COMM SMOVL C00306 BC00306 V=60.0  +MOVJ EC00306
COMM SMOVL C00307 BC00307 V=60.0  +MOVJ EC00307
COMM SREFP 3 C00308 BC00308  +REFP EC00308
COMM CALL JOB:SEARCH-R1-S13D
COMM SET P041 P006
COMM SFTON3D P041
COMM SMOVL C00309 BC00309 V=60.0  +MOVJ EC00309
COMM MOVL C00310 BC00310 V=400.0  +MOVJ EC00310 VJ=100.00
COMM MOVL C00311 BC00311 V=1000.0  +MOVJ EC00311 VJ=100.00
COMM 'Path S1858
COMM SFTOF3D
COMM MOVJ C00312 BC00312 VJ=100.00  +MOVJ EC00312 VJ=100.00
COMM MOVL C00313 BC00313 V=400.0  +MOVJ EC00313 VJ=100.00
COMM SMOVL C00314 BC00314 V=60.0  +MOVJ EC00314
COMM SREFP 3 C00315 BC00315  +REFP EC00315
COMM CALL JOB:SEARCH-R1-S13D
COMM SET P040 P006
COMM SFTON3D P040
COMM SMOVL C00316 BC00316 V=60.0  +MOVJ EC00316
COMM SMOVL C00317 BC00317 V=60.0  +MOVJ EC00317
COMM SREFP 3 C00318 BC00318  +REFP EC00318
COMM CALL JOB:SEARCH-R1-S13D
COMM SET P040 P006
COMM SFTON3D P040
COMM SMOVL C00319 BC00319 V=60.0  +MOVJ EC00319
COMM MOVL C00320 BC00320 V=400.0  +MOVJ EC00320 VJ=100.00
COMM MOVL C00321 BC00321 V=1000.0  +MOVJ EC00321 VJ=100.00
MOVL C00322 BC00322 V=1000.0  +MOVJ EC00322 VJ=100.00
'Path S1859
SFTOF3D
MOVJ C00323 BC00323 VJ=100.00  +MOVJ EC00323 VJ=100.00
MOVJ C00324 BC00324 VJ=100.00  +MOVJ EC00324 VJ=100.00
MOVL C00325 BC00325 V=400.0  +MOVJ EC00325 VJ=100.00
SMOVL C00326 BC00326 V=60.0  +MOVJ EC00326
SREFP 3 C00327 BC00327  +REFP EC00327
CALL JOB:SEARCH-R1-S13D
SET P043 P006
SFTON3D P043
SMOVL C00328 BC00328 V=60.0  +MOVJ EC00328
SMOVL C00329 BC00329 V=60.0  +MOVJ EC00329
SREFP 3 C00330 BC00330  +REFP EC00330
CALL JOB:SEARCH-R1-S13D
SET P043 P006
SFTON3D P043
SMOVL C00331 BC00331 V=60.0  +MOVJ EC00331
MOVL C00332 BC00332 V=400.0  +MOVJ EC00332 VJ=100.00
MOVL C00333 BC00333 V=1000.0  +MOVJ EC00333 VJ=100.00
'Path S1860
SFTOF3D
MOVJ C00334 BC00334 VJ=100.00  +MOVJ EC00334 VJ=100.00
MOVL C00335 BC00335 V=400.0  +MOVJ EC00335 VJ=100.00
SMOVL C00336 BC00336 V=60.0  +MOVJ EC00336
SREFP 3 C00337 BC00337  +REFP EC00337
CALL JOB:SEARCH-R1-S13D
SET P039 P006
SFTON3D P039
SMOVL C00338 BC00338 V=60.0  +MOVJ EC00338
SMOVL C00339 BC00339 V=60.0  +MOVJ EC00339
SREFP 3 C00340 BC00340  +REFP EC00340
CALL JOB:SEARCH-R1-S13D
SET P039 P006
SFTON3D P039
SMOVL C00341 BC00341 V=60.0  +MOVJ EC00341
MOVL C00342 BC00342 V=400.0  +MOVJ EC00342 VJ=100.00
MOVL C00343 BC00343 V=1000.0  +MOVJ EC00343 VJ=100.00
MOVJ C00344 BC00344 VJ=100.00  +MOVJ EC00344 VJ=100.00
'Path S1861
SFTOF3D
MOVJ C00345 BC00345 VJ=100.00  +MOVJ EC00345 VJ=100.00
MOVL C00346 BC00346 V=400.0  +MOVJ EC00346 VJ=100.00
SMOVL C00347 BC00347 V=60.0  +MOVJ EC00347
SREFP 3 C00348 BC00348  +REFP EC00348
CALL JOB:SEARCH-R1-S13D
SET P034 P006
SFTON3D P034
SMOVL C00349 BC00349 V=60.0  +MOVJ EC00349
SMOVL C00350 BC00350 V=60.0  +MOVJ EC00350
SREFP 3 C00351 BC00351  +REFP EC00351
CALL JOB:SEARCH-R1-S13D
SET P034 P006
SFTON3D P034
SMOVL C00352 BC00352 V=60.0  +MOVJ EC00352
MOVL C00353 BC00353 V=400.0  +MOVJ EC00353 VJ=100.00
MOVL C00354 BC00354 V=1000.0  +MOVJ EC00354 VJ=100.00
MOVJ C00355 BC00355 VJ=100.00  +MOVJ EC00355 VJ=100.00
'Path S1862
SFTOF3D
MOVJ C00356 BC00356 VJ=100.00  +MOVJ EC00356 VJ=100.00
MOVL C00357 BC00357 V=400.0  +MOVJ EC00357 VJ=100.00
SMOVL C00358 BC00358 V=60.0  +MOVJ EC00358
SREFP 3 C00359 BC00359  +REFP EC00359
CALL JOB:SEARCH-R1-S13D
SET P038 P006
SFTON3D P038
SMOVL C00360 BC00360 V=60.0  +MOVJ EC00360
SMOVL C00361 BC00361 V=60.0  +MOVJ EC00361
SREFP 3 C00362 BC00362  +REFP EC00362
CALL JOB:SEARCH-R1-S13D
SET P038 P006
SFTON3D P038
SMOVL C00363 BC00363 V=60.0  +MOVJ EC00363
SMOVL C00364 BC00364 V=60.0  +MOVJ EC00364
SREFP 3 C00365 BC00365  +REFP EC00365
CALL JOB:SEARCH-R1-S13D
SET P038 P006
SFTON3D P038
SMOVL C00366 BC00366 V=60.0  +MOVJ EC00366
MOVL C00367 BC00367 V=400.0  +MOVJ EC00367 VJ=100.00
MOVL C00368 BC00368 V=1000.0  +MOVJ EC00368 VJ=100.00
'Path S1863
SFTOF3D
MOVJ C00369 BC00369 VJ=100.00  +MOVJ EC00369 VJ=100.00
MOVL C00370 BC00370 V=400.0  +MOVJ EC00370 VJ=100.00
SMOVL C00371 BC00371 V=60.0  +MOVJ EC00371
SREFP 3 C00372 BC00372  +REFP EC00372
CALL JOB:SEARCH-R1-S13D
SET P033 P006
SFTON3D P033
SMOVL C00373 BC00373 V=60.0  +MOVJ EC00373
SMOVL C00374 BC00374 V=60.0  +MOVJ EC00374
SREFP 3 C00375 BC00375  +REFP EC00375
CALL JOB:SEARCH-R1-S13D
SET P033 P006
SFTON3D P033
SMOVL C00376 BC00376 V=60.0  +MOVJ EC00376
MOVL C00377 BC00377 V=400.0  +MOVJ EC00377 VJ=100.00
MOVL C00378 BC00378 V=1000.0  +MOVJ EC00378 VJ=100.00
MOVL C00379 BC00379 V=1000.0  +MOVJ EC00379 VJ=100.00
'Path S1864
SFTOF3D
MOVJ C00380 BC00380 VJ=100.00  +MOVJ EC00380 VJ=100.00
MOVJ C00381 BC00381 VJ=100.00  +MOVJ EC00381 VJ=100.00
MOVL C00382 BC00382 V=400.0  +MOVJ EC00382 VJ=100.00
SMOVL C00383 BC00383 V=60.0  +MOVJ EC00383
SREFP 3 C00384 BC00384  +REFP EC00384
CALL JOB:SEARCH-R1-S13D
SET P035 P006
SFTON3D P035
SMOVL C00385 BC00385 V=60.0  +MOVJ EC00385
SMOVL C00386 BC00386 V=60.0  +MOVJ EC00386
SREFP 3 C00387 BC00387  +REFP EC00387
CALL JOB:SEARCH-R1-S13D
SET P035 P006
SFTON3D P035
SMOVL C00388 BC00388 V=60.0  +MOVJ EC00388
MOVL C00389 BC00389 V=400.0  +MOVJ EC00389 VJ=100.00
MOVL C00390 BC00390 V=1000.0  +MOVJ EC00390 VJ=100.00
MOVL C00391 BC00391 V=1000.0  +MOVJ EC00391 VJ=100.00
'Path S1865
SFTOF3D
MOVJ C00392 BC00392 VJ=100.00  +MOVJ EC00392 VJ=100.00
MOVL C00393 BC00393 V=400.0  +MOVJ EC00393 VJ=100.00
SMOVL C00394 BC00394 V=60.0  +MOVJ EC00394
SREFP 3 C00395 BC00395  +REFP EC00395
CALL JOB:SEARCH-R1-S13D
SET P037 P006
SFTON3D P037
SMOVL C00396 BC00396 V=60.0  +MOVJ EC00396
SMOVL C00397 BC00397 V=60.0  +MOVJ EC00397
SREFP 3 C00398 BC00398  +REFP EC00398
CALL JOB:SEARCH-R1-S13D
SET P037 P006
SFTON3D P037
SMOVL C00399 BC00399 V=60.0  +MOVJ EC00399
MOVL C00400 BC00400 V=400.0  +MOVJ EC00400 VJ=100.00
MOVL C00401 BC00401 V=1000.0  +MOVJ EC00401 VJ=100.00
'Path S1866
SFTOF3D
MOVJ C00402 BC00402 VJ=100.00  +MOVJ EC00402 VJ=100.00
MOVJ C00403 BC00403 VJ=100.00  +MOVJ EC00403 VJ=100.00
MOVL C00404 BC00404 V=400.0  +MOVJ EC00404 VJ=100.00
SMOVL C00405 BC00405 V=60.0  +MOVJ EC00405
SREFP 3 C00406 BC00406  +REFP EC00406
CALL JOB:SEARCH-R1-S13D
SET P031 P006
SFTON3D P031
SMOVL C00407 BC00407 V=60.0  +MOVJ EC00407
SMOVL C00408 BC00408 V=60.0  +MOVJ EC00408
SREFP 3 C00409 BC00409  +REFP EC00409
CALL JOB:SEARCH-R1-S13D
SET P031 P006
SFTON3D P031
SMOVL C00410 BC00410 V=60.0  +MOVJ EC00410
MOVL C00411 BC00411 V=400.0  +MOVJ EC00411 VJ=100.00
MOVL C00412 BC00412 V=1000.0  +MOVJ EC00412 VJ=100.00
'Path S1867
MOVJ C00413 BC00413 VJ=20.00  +MOVJ EC00413 VJ=20.00
MOVJ C00414 BC00414 VJ=20.00  +MOVJ EC00414 VJ=20.00
SFTOF3D
MOVJ C00415 BC00415 VJ=100.00  +MOVJ EC00415 VJ=100.00
MOVL C00416 BC00416 V=400.0  +MOVJ EC00416 VJ=100.00
SMOVL C00417 BC00417 V=60.0  +MOVJ EC00417
SREFP 3 C00418 BC00418  +REFP EC00418
CALL JOB:SEARCH-R1-S13D
SET P036 P006
SFTON3D P036
SMOVL C00419 BC00419 V=60.0  +MOVJ EC00419
SMOVL C00420 BC00420 V=60.0  +MOVJ EC00420
SREFP 3 C00421 BC00421  +REFP EC00421
CALL JOB:SEARCH-R1-S13D
SET P036 P006
SFTON3D P036
SMOVL C00422 BC00422 V=60.0  +MOVJ EC00422
MOVL C00423 BC00423 V=400.0  +MOVJ EC00423 VJ=100.00
MOVL C00424 BC00424 V=1000.0  +MOVJ EC00424 VJ=100.00
MOVL C00425 BC00425 V=1000.0  +MOVJ EC00425 VJ=100.00
'Path S1868
SFTOF3D
MOVJ C00426 BC00426 VJ=100.00  +MOVJ EC00426 VJ=100.00
MOVL C00427 BC00427 V=400.0  +MOVJ EC00427 VJ=100.00
SMOVL C00428 BC00428 V=60.0  +MOVJ EC00428
SREFP 3 C00429 BC00429  +REFP EC00429
CALL JOB:SEARCH-R1-S13D
SET P032 P006
SFTON3D P032
SMOVL C00430 BC00430 V=60.0  +MOVJ EC00430
SMOVL C00431 BC00431 V=60.0  +MOVJ EC00431
SREFP 3 C00432 BC00432  +REFP EC00432
CALL JOB:SEARCH-R1-S13D
SET P032 P006
SFTON3D P032
SMOVL C00433 BC00433 V=60.0  +MOVJ EC00433
MOVL C00434 BC00434 V=400.0  +MOVJ EC00434 VJ=100.00
MOVL C00435 BC00435 V=1000.0  +MOVJ EC00435 VJ=100.00
'Path W1869
SFTOF3D
SFTON3D P032
MOVJ C00436 BC00436 VJ=100.00  +MOVJ EC00436 VJ=100.00
SMOVL C00437 BC00437 V=400.0  +MOVJ EC00437
SMOVL C00438 BC00438 V=100.0 PL=0  +MOVJ EC00438
SREFP 1 C00439 BC00439  +REFP EC00439
SREFP 2 C00440 BC00440  +REFP EC00440
MACRO1 MJ#(0) ARGF0
ARCON
SMOVL C00441 BC00441 V=10.0  +MOVJ EC00441
SMOVL C00442 BC00442 V=10.0  +MOVJ EC00442
SMOVL C00443 BC00443 V=10.0  +MOVJ EC00443
ARCOF
SMOVL C00444 BC00444 V=400.0  +MOVJ EC00444
SMOVL C00445 BC00445 V=1000.0  +MOVJ EC00445
SMOVL C00446 BC00446 V=1000.0  +MOVJ EC00446
SFTOF3D
MOVJ C00447 BC00447 VJ=100.00  +MOVJ EC00447 VJ=100.00
'Path W1870
SFTOF3D
SFTON3D P033
MOVJ C00448 BC00448 VJ=100.00  +MOVJ EC00448 VJ=100.00
MOVJ C00449 BC00449 VJ=100.00  +MOVJ EC00449 VJ=100.00
SMOVL C00450 BC00450 V=400.0  +MOVJ EC00450
SMOVL C00451 BC00451 V=100.0 PL=0  +MOVJ EC00451
SREFP 1 C00452 BC00452  +REFP EC00452
SREFP 2 C00453 BC00453  +REFP EC00453
MACRO1 MJ#(0) ARGF0
ARCON
SMOVL C00454 BC00454 V=10.0  +MOVJ EC00454
SMOVL C00455 BC00455 V=10.0  +MOVJ EC00455
SMOVL C00456 BC00456 V=10.0  +MOVJ EC00456
ARCOF
SMOVL C00457 BC00457 V=400.0  +MOVJ EC00457
SMOVL C00458 BC00458 V=1000.0  +MOVJ EC00458
SFTOF3D
'Path W1871
SFTOF3D
SFTON3D P034
MOVJ C00459 BC00459 VJ=100.00  +MOVJ EC00459 VJ=100.00
SMOVL C00460 BC00460 V=400.0  +MOVJ EC00460
SMOVL C00461 BC00461 V=100.0 PL=0  +MOVJ EC00461
SREFP 1 C00462 BC00462  +REFP EC00462
SREFP 2 C00463 BC00463  +REFP EC00463
MACRO1 MJ#(0) ARGF0
ARCON
SMOVL C00464 BC00464 V=10.0  +MOVJ EC00464
SMOVL C00465 BC00465 V=10.0  +MOVJ EC00465
ARCOF
SMOVL C00466 BC00466 V=400.0  +MOVJ EC00466
SMOVL C00467 BC00467 V=1000.0  +MOVJ EC00467
SMOVL C00468 BC00468 V=1000.0  +MOVJ EC00468
SFTOF3D
MOVJ C00469 BC00469 VJ=20.00  +MOVJ EC00469 VJ=20.00
MOVJ C00470 BC00470 VJ=20.00  +MOVJ EC00470 VJ=20.00
'Path W1872
SFTOF3D
SFTON3D P031
MOVJ C00471 BC00471 VJ=100.00  +MOVJ EC00471 VJ=100.00
SMOVL C00472 BC00472 V=400.0  +MOVJ EC00472
SMOVL C00473 BC00473 V=100.0 PL=0  +MOVJ EC00473
SREFP 1 C00474 BC00474  +REFP EC00474
SREFP 2 C00475 BC00475  +REFP EC00475
MACRO1 MJ#(0) ARGF0
ARCON
SMOVL C00476 BC00476 V=10.0  +MOVJ EC00476
SMOVL C00477 BC00477 V=10.0  +MOVJ EC00477
ARCOF
SMOVL C00478 BC00478 V=400.0  +MOVJ EC00478
SMOVL C00479 BC00479 V=1000.0  +MOVJ EC00479
SMOVL C00480 BC00480 V=1000.0  +MOVJ EC00480
SFTOF3D
'Path W1873
MOVJ C00481 BC00481 VJ=20.00  +MOVJ EC00481 VJ=20.00
SFTOF3D
SFTON3D P035
MOVJ C00482 BC00482 VJ=100.00  +MOVJ EC00482 VJ=100.00
SMOVL C00483 BC00483 V=400.0  +MOVJ EC00483
SMOVL C00484 BC00484 V=100.0 PL=0  +MOVJ EC00484
SREFP 1 C00485 BC00485  +REFP EC00485
SREFP 2 C00486 BC00486  +REFP EC00486
MACRO1 MJ#(0) ARGF0
ARCON
SMOVL C00487 BC00487 V=10.0  +MOVJ EC00487
SMOVL C00488 BC00488 V=10.0  +MOVJ EC00488
ARCOF
SMOVL C00489 BC00489 V=400.0  +MOVJ EC00489
SMOVL C00490 BC00490 V=1000.0  +MOVJ EC00490
SMOVL C00491 BC00491 V=1000.0  +MOVJ EC00491
SFTOF3D
MOVJ C00492 BC00492 VJ=100.00  +MOVJ EC00492 VJ=100.00
'Path W1874
SFTOF3D
SFTON3D P036
MOVJ C00493 BC00493 VJ=100.00  +MOVJ EC00493 VJ=100.00
SMOVL C00494 BC00494 V=400.0  +MOVJ EC00494
SMOVL C00495 BC00495 V=100.0 PL=0  +MOVJ EC00495
SREFP 1 C00496 BC00496  +REFP EC00496
SREFP 2 C00497 BC00497  +REFP EC00497
MACRO1 MJ#(0) ARGF0
ARCON
SMOVL C00498 BC00498 V=10.0  +MOVJ EC00498
SMOVL C00499 BC00499 V=10.0  +MOVJ EC00499
SMOVL C00500 BC00500 V=10.0  +MOVJ EC00500
ARCOF
SMOVL C00501 BC00501 V=400.0  +MOVJ EC00501
SMOVL C00502 BC00502 V=1000.0  +MOVJ EC00502
SMOVL C00503 BC00503 V=1000.0  +MOVJ EC00503
SFTOF3D
MOVJ C00504 BC00504 VJ=100.00  +MOVJ EC00504 VJ=100.00
'Path W1875
SFTOF3D
SFTON3D P037
MOVJ C00505 BC00505 VJ=100.00  +MOVJ EC00505 VJ=100.00
MOVJ C00506 BC00506 VJ=100.00  +MOVJ EC00506 VJ=100.00
SMOVL C00507 BC00507 V=400.0  +MOVJ EC00507
SMOVL C00508 BC00508 V=100.0 PL=0  +MOVJ EC00508
SREFP 1 C00509 BC00509  +REFP EC00509
SREFP 2 C00510 BC00510  +REFP EC00510
MACRO1 MJ#(0) ARGF0
ARCON
SMOVL C00511 BC00511 V=10.0  +MOVJ EC00511
SMOVL C00512 BC00512 V=10.0  +MOVJ EC00512
SMOVL C00513 BC00513 V=10.0  +MOVJ EC00513
ARCOF
SMOVL C00514 BC00514 V=400.0  +MOVJ EC00514
SMOVL C00515 BC00515 V=1000.0  +MOVJ EC00515
SMOVL C00516 BC00516 V=1000.0  +MOVJ EC00516
SFTOF3D
MOVJ C00517 BC00517 VJ=100.00  +MOVJ EC00517 VJ=100.00
'Path W1876
SFTOF3D
SFTON3D P038
MOVJ C00518 BC00518 VJ=100.00  +MOVJ EC00518 VJ=100.00
MOVJ C00519 BC00519 VJ=100.00  +MOVJ EC00519 VJ=100.00
SMOVL C00520 BC00520 V=400.0  +MOVJ EC00520
SMOVL C00521 BC00521 V=100.0 PL=0  +MOVJ EC00521
SREFP 1 C00522 BC00522  +REFP EC00522
SREFP 2 C00523 BC00523  +REFP EC00523
MACRO1 MJ#(0) ARGF0
ARCON
SMOVL C00524 BC00524 V=10.0  +MOVJ EC00524
SMOVL C00525 BC00525 V=10.0  +MOVJ EC00525
ARCOF
SMOVL C00526 BC00526 V=400.0  +MOVJ EC00526
SMOVL C00527 BC00527 V=1000.0  +MOVJ EC00527
SFTOF3D
'Path W1877
SFTOF3D
SFTON3D P038
SMOVL C00528 BC00528 V=400.0  +MOVJ EC00528
SMOVL C00529 BC00529 V=100.0 PL=0  +MOVJ EC00529
SREFP 1 C00530 BC00530  +REFP EC00530
SREFP 2 C00531 BC00531  +REFP EC00531
MACRO1 MJ#(0) ARGF0
ARCON
SMOVL C00532 BC00532 V=10.0  +MOVJ EC00532
SMOVL C00533 BC00533 V=10.0  +MOVJ EC00533
SMOVL C00534 BC00534 V=10.0  +MOVJ EC00534
ARCOF
SMOVL C00535 BC00535 V=400.0  +MOVJ EC00535
SFTOF3D
MOVJ C00536 BC00536 VJ=100.00  +MOVJ EC00536 VJ=100.00
'Path W1878
SFTOF3D
SFTON3D P039
MOVJ C00537 BC00537 VJ=100.00  +MOVJ EC00537 VJ=100.00
MOVJ C00538 BC00538 VJ=100.00  +MOVJ EC00538 VJ=100.00
SMOVL C00539 BC00539 V=400.0  +MOVJ EC00539
SMOVL C00540 BC00540 V=100.0 PL=0  +MOVJ EC00540
SREFP 1 C00541 BC00541  +REFP EC00541
SREFP 2 C00542 BC00542  +REFP EC00542
MACRO1 MJ#(0) ARGF0
ARCON
SMOVL C00543 BC00543 V=10.0  +MOVJ EC00543
ARCOF
SMOVL C00544 BC00544 V=400.0  +MOVJ EC00544
SMOVL C00545 BC00545 V=1000.0  +MOVJ EC00545
SMOVL C00546 BC00546 V=1000.0  +MOVJ EC00546
SFTOF3D
'Path W1879
SFTOF3D
SFTON3D P042
MOVJ C00547 BC00547 VJ=100.00  +MOVJ EC00547 VJ=100.00
COMM MOVJ C00548 BC00548 VJ=100.00  +MOVJ EC00548 VJ=100.00
COMM SMOVL C00549 BC00549 V=400.0  +MOVJ EC00549
COMM SMOVL C00550 BC00550 V=100.0 PL=0  +MOVJ EC00550
COMM SREFP 1 C00551 BC00551  +REFP EC00551
COMM SREFP 2 C00552 BC00552  +REFP EC00552
COMM MACRO1 MJ#(0) ARGF0
COMM ARCON
COMM SMOVL C00553 BC00553 V=10.0  +MOVJ EC00553
COMM SMOVL C00554 BC00554 V=10.0  +MOVJ EC00554
COMM SMOVL C00555 BC00555 V=10.0  +MOVJ EC00555
COMM ARCOF
COMM SMOVL C00556 BC00556 V=400.0  +MOVJ EC00556
COMM SMOVL C00557 BC00557 V=1000.0  +MOVJ EC00557
SFTOF3D
'Path W1880
COMM SFTOF3D
COMM SFTON3D P041
COMM MOVJ C00558 BC00558 VJ=100.00  +MOVJ EC00558 VJ=100.00
COMM SMOVL C00559 BC00559 V=400.0  +MOVJ EC00559
COMM SMOVL C00560 BC00560 V=100.0 PL=0  +MOVJ EC00560
COMM SREFP 1 C00561 BC00561  +REFP EC00561
COMM SREFP 2 C00562 BC00562  +REFP EC00562
COMM MACRO1 MJ#(0) ARGF0
COMM ARCON
COMM SMOVL C00563 BC00563 V=10.0  +MOVJ EC00563
COMM ARCOF
COMM SMOVL C00564 BC00564 V=400.0  +MOVJ EC00564
COMM SMOVL C00565 BC00565 V=1000.0  +MOVJ EC00565
SFTOF3D
'Path W1881
COMM SFTOF3D
COMM SFTON3D P040
COMM MOVJ C00566 BC00566 VJ=100.00  +MOVJ EC00566 VJ=100.00
COMM SMOVL C00567 BC00567 V=400.0  +MOVJ EC00567
COMM SMOVL C00568 BC00568 V=100.0 PL=0  +MOVJ EC00568
COMM SREFP 1 C00569 BC00569  +REFP EC00569
COMM SREFP 2 C00570 BC00570  +REFP EC00570
COMM MACRO1 MJ#(0) ARGF0
COMM ARCON
COMM SMOVL C00571 BC00571 V=10.0  +MOVJ EC00571
COMM ARCOF
COMM SMOVL C00572 BC00572 V=400.0  +MOVJ EC00572
COMM SMOVL C00573 BC00573 V=1000.0  +MOVJ EC00573
COMM SMOVL C00574 BC00574 V=1000.0  +MOVJ EC00574
SFTOF3D
MOVJ C00575 BC00575 VJ=20.00  +MOVJ EC00575 VJ=20.00
'Path W1882
SFTOF3D
SFTON3D P043
MOVJ C00576 BC00576 VJ=100.00  +MOVJ EC00576 VJ=100.00
SMOVL C00577 BC00577 V=400.0  +MOVJ EC00577
SMOVL C00578 BC00578 V=100.0 PL=0  +MOVJ EC00578
SREFP 1 C00579 BC00579  +REFP EC00579
SREFP 2 C00580 BC00580  +REFP EC00580
MACRO1 MJ#(0) ARGF0
ARCON
COMM SMOVL C00581 BC00581 V=10.0  +MOVJ EC00581
COMM SMOVL C00582 BC00582 V=10.0  +MOVJ EC00582
COMM SMOVL C00583 BC00583 V=10.0  +MOVJ EC00583
COMM SMOVL C00584 BC00584 V=10.0  +MOVJ EC00584
COMM SMOVL C00585 BC00585 V=10.0  +MOVJ EC00585
COMM SMOVL C00586 BC00586 V=10.0  +MOVJ EC00586
COMM SMOVL C00587 BC00587 V=10.0  +MOVJ EC00587
SMOVL C00588 BC00588 V=10.0  +MOVJ EC00588
SMOVL C00589 BC00589 V=10.0  +MOVJ EC00589
SMOVL C00590 BC00590 V=10.0  +MOVJ EC00590
SMOVL C00591 BC00591 V=10.0  +MOVJ EC00591
SMOVL C00592 BC00592 V=10.0  +MOVJ EC00592
SMOVL C00593 BC00593 V=10.0  +MOVJ EC00593
SMOVL C00594 BC00594 V=10.0  +MOVJ EC00594
SMOVL C00595 BC00595 V=10.0  +MOVJ EC00595
ARCOF
SMOVL C00596 BC00596 V=400.0  +MOVJ EC00596
SMOVL C00597 BC00597 V=1000.0  +MOVJ EC00597
SFTOF3D
MOVJ C00598 BC00598 VJ=100.00  +MOVJ EC00598 VJ=100.00
MOVJ C00599 BC00599 VJ=100.00  +MOVJ EC00599 VJ=100.00
MOVJ C00600 BC00600 VJ=100.00  +MOVJ EC00600 VJ=100.00
*LABEL
MOVJ C00601 BC00601 VJ=50.00  +MOVJ EC00601 VJ=20.00
MOVJ C00602 BC00602 VJ=100.00  +MOVJ EC00602 VJ=100.00
MOVJ C00603 BC00603 VJ=100.00  +MOVJ EC00603 VJ=100.00
'1
'BRAKUJACY ELEMENT
'BRAKUJACY ELEMENT
'BRAKUJACY ELEMENT
'Path W1886
COMM SFTOF3D
COMM SFTON3D P023
COMM MOVJ C00604 BC00604 VJ=100.00  +MOVJ EC00604 VJ=100.00
COMM SMOVL C00605 BC00605 V=400.0  +MOVJ EC00605
COMM SMOVL C00606 BC00606 V=100.0 PL=0  +MOVJ EC00606
COMM SREFP 1 C00607 BC00607  +REFP EC00607
COMM SREFP 2 C00608 BC00608  +REFP EC00608
COMM MACRO1 MJ#(0) ARGF0
COMM ARCON
COMM SMOVL C00609 BC00609 V=10.0  +MOVJ EC00609
COMM SMOVL C00610 BC00610 V=10.0  +MOVJ EC00610
COMM SMOVL C00611 BC00611 V=10.0  +MOVJ EC00611
COMM ARCOF
COMM SMOVL C00612 BC00612 V=400.0  +MOVJ EC00612
COMM SMOVL C00613 BC00613 V=1000.0  +MOVJ EC00613
COMM SFTOF3D
'Path W1887
SFTOF3D
SFTON3D P023
MOVJ C00614 BC00614 VJ=100.00  +MOVJ EC00614 VJ=100.00
SMOVL C00615 BC00615 V=400.0  +MOVJ EC00615
SMOVL C00616 BC00616 V=100.0 PL=0  +MOVJ EC00616
SREFP 1 C00617 BC00617  +REFP EC00617
SREFP 2 C00618 BC00618  +REFP EC00618
MACRO1 MJ#(0) ARGF9
ARCON
SMOVL C00619 BC00619 V=10.0  +MOVJ EC00619
ARCOF
SMOVL C00620 BC00620 V=400.0  +MOVJ EC00620
SMOVL C00621 BC00621 V=1000.0  +MOVJ EC00621
SFTOF3D
MOVJ C00622 BC00622 VJ=100.00  +MOVJ EC00622 VJ=100.00
MOVJ C00623 BC00623 VJ=100.00  +MOVJ EC00623 VJ=100.00
MOVJ C00624 BC00624 VJ=100.00  +MOVJ EC00624 VJ=100.00
'2
MOVJ C00625 BC00625 VJ=100.00  +MOVJ EC00625 VJ=100.00
MOVJ C00626 BC00626 VJ=100.00  +MOVJ EC00626 VJ=20.00
MOVJ C00627 BC00627 VJ=100.00  +MOVJ EC00627 VJ=100.00
'Path W1888
SFTOF3D
SFTON3D P021
MOVJ C00628 BC00628 VJ=15.00  +MOVJ EC00628 VJ=100.00
SMOVL C00629 BC00629 V=400.0  +MOVJ EC00629
SMOVL C00630 BC00630 V=133.3 PL=0  +MOVJ EC00630
SREFP 1 C00631 BC00631  +REFP EC00631
SREFP 2 C00632 BC00632  +REFP EC00632
MACRO1 MJ#(0) ARGF14
ARCON
SMOVL C00633 BC00633 V=10.0  +MOVJ EC00633
ARCOF
SMOVL C00634 BC00634 V=166.7  +MOVJ EC00634
SMOVL C00635 BC00635 V=166.7  +MOVJ EC00635
MACRO1 MJ#(0) ARGF14
SMOVL C00636 BC00636 V=133.3 PL=0  +MOVJ EC00636
ARCON
SMOVL C00637 BC00637 V=10.0  +MOVJ EC00637
ARCOF
SMOVL C00638 BC00638 V=400.0  +MOVJ EC00638
SMOVL C00639 BC00639 V=1000.0  +MOVJ EC00639
SMOVL C00640 BC00640 V=1000.0  +MOVJ EC00640
SFTOF3D
MOVJ C00641 BC00641 VJ=50.00  +MOVJ EC00641 VJ=20.00
MOVJ C00642 BC00642 VJ=100.00  +MOVJ EC00642 VJ=100.00
'Path W1889
SFTOF3D
SFTON3D P021
MOVJ C00643 BC00643 VJ=100.00  +MOVJ EC00643 VJ=100.00
MOVJ C00644 BC00644 VJ=100.00  +MOVJ EC00644 VJ=100.00
SMOVL C00645 BC00645 V=400.0  +MOVJ EC00645
SMOVL C00646 BC00646 V=133.3 PL=0  +MOVJ EC00646
SREFP 1 C00647 BC00647  +REFP EC00647
SREFP 2 C00648 BC00648  +REFP EC00648
MACRO1 MJ#(0) ARGF14
ARCON
SMOVL C00649 BC00649 V=10.0  +MOVJ EC00649
ARCOF
SMOVL C00650 BC00650 V=166.7  +MOVJ EC00650
SMOVL C00651 BC00651 V=166.7  +MOVJ EC00651
SMOVL C00652 BC00652 V=166.7 PL=0  +MOVJ EC00652
ARCON
SMOVL C00653 BC00653 V=10.0  +MOVJ EC00653
ARCOF
SMOVL C00654 BC00654 V=400.0  +MOVJ EC00654
SMOVL C00655 BC00655 V=1000.0  +MOVJ EC00655
SMOVL C00656 BC00656 V=1000.0  +MOVJ EC00656
SFTOF3D
MOVL C00657 BC00657 V=400.0  +MOVJ EC00657 VJ=100.00
MOVJ C00658 BC00658 VJ=100.00  +MOVJ EC00658 VJ=100.00
MOVL C00659 BC00659 V=666.7  +MOVJ EC00659 VJ=100.00
SFTON3D P050
MACRO1 MJ#(0) ARGF9
SMOVL C00660 BC00660 V=400.0  +MOVJ EC00660
SMOVL C00661 BC00661 V=150.0 PL=0  +MOVJ EC00661
ARCON
SFTON3D P051
SMOVL C00662 BC00662 V=11.7  +MOVJ EC00662
SMOVC C00663 BC00663 V=13.3  +MOVJ EC00663
SMOVC C00664 BC00664 V=13.3  +MOVJ EC00664
SMOVC C00665 BC00665 V=13.3  +MOVJ EC00665
SFTON3D P050
SMOVL C00666 BC00666 V=11.7  +MOVJ EC00666
SMOVL C00667 BC00667 V=11.7  +MOVJ EC00667
SMOVC C00668 BC00668 V=13.3  +MOVJ EC00668
SMOVC C00669 BC00669 V=13.3  +MOVJ EC00669
SMOVC C00670 BC00670 V=13.3  +MOVJ EC00670
ARCOF
SMOVL C00671 BC00671 V=333.3  +MOVJ EC00671
SFTOF3D
MOVJ C00672 BC00672 VJ=100.00  +MOVJ EC00672 VJ=20.00
MOVJ C00673 BC00673 VJ=100.00  +MOVJ EC00673 VJ=100.00
MOVJ C00674 BC00674 VJ=100.00  +MOVJ EC00674 VJ=100.00
MOVJ C00675 BC00675 VJ=100.00  +MOVJ EC00675 VJ=100.00
MOVJ C00676 BC00676 VJ=100.00  +MOVJ EC00676 VJ=100.00
'3
'Path W1890
SFTOF3D
SFTON3D P023
MOVJ C00677 BC00677 VJ=100.00  +MOVJ EC00677 VJ=100.00
'BRAKUJACY ELEMENT
COMM SMOVL C00678 BC00678 V=400.0  +MOVJ EC00678
COMM SMOVL C00679 BC00679 V=100.0 PL=0  +MOVJ EC00679
COMM SREFP 1 C00680 BC00680  +REFP EC00680
COMM SREFP 2 C00681 BC00681  +REFP EC00681
COMM MACRO1 MJ#(0) ARGF0
COMM ARCON
COMM SMOVL C00682 BC00682 V=10.0  +MOVJ EC00682
COMM SMOVL C00683 BC00683 V=10.0  +MOVJ EC00683
COMM SMOVL C00684 BC00684 V=10.0  +MOVJ EC00684
COMM ARCOF
COMM SMOVL C00685 BC00685 V=400.0  +MOVJ EC00685
COMM SMOVL C00686 BC00686 V=1000.0  +MOVJ EC00686
SFTOF3D
'Path W1891
SFTOF3D
SFTON3D P023
MOVJ C00687 BC00687 VJ=100.00  +MOVJ EC00687 VJ=100.00
SMOVL C00688 BC00688 V=400.0  +MOVJ EC00688
SMOVL C00689 BC00689 V=133.3 PL=0  +MOVJ EC00689
SREFP 1 C00690 BC00690  +REFP EC00690
SREFP 2 C00691 BC00691  +REFP EC00691
MACRO1 MJ#(0) ARGF14
ARCON
SMOVL C00692 BC00692 V=11.7  +MOVJ EC00692
ARCOF
SMOVL C00693 BC00693 V=400.0  +MOVJ EC00693
SMOVL C00694 BC00694 V=1000.0  +MOVJ EC00694
SFTOF3D
MOVJ C00695 BC00695 VJ=100.00  +MOVJ EC00695 VJ=100.00
MOVJ C00696 BC00696 VJ=100.00  +MOVJ EC00696 VJ=20.00
MOVJ C00697 BC00697 VJ=100.00  +MOVJ EC00697 VJ=100.00
MOVJ C00698 BC00698 VJ=100.00  +MOVJ EC00698 VJ=20.00
MOVJ C00699 BC00699 VJ=100.00  +MOVJ EC00699 VJ=100.00
MOVJ C00700 BC00700 VJ=100.00  +MOVJ EC00700 VJ=100.00
'4
'Path W1892
SFTOF3D
SFTON3D P021
MOVJ C00701 BC00701 VJ=100.00  +MOVJ EC00701 VJ=20.00
SMOVL C00702 BC00702 V=400.0  +MOVJ EC00702
SMOVL C00703 BC00703 V=133.3 PL=0  +MOVJ EC00703
SREFP 1 C00704 BC00704  +REFP EC00704
SREFP 2 C00705 BC00705  +REFP EC00705
MACRO1 MJ#(0) ARGF14
ARCON
SMOVL C00706 BC00706 V=10.0  +MOVJ EC00706
ARCOF
SMOVL C00707 BC00707 V=400.0  +MOVJ EC00707
SMOVL C00708 BC00708 V=1000.0  +MOVJ EC00708
SFTOF3D
'Path W1893
SFTOF3D
SFTON3D P021
MOVJ C00709 BC00709 VJ=20.00  +MOVJ EC00709 VJ=100.00
SMOVL C00710 BC00710 V=400.0  +MOVJ EC00710
SMOVL C00711 BC00711 V=133.3 PL=0  +MOVJ EC00711
SREFP 1 C00712 BC00712  +REFP EC00712
SREFP 2 C00713 BC00713  +REFP EC00713
MACRO1 MJ#(0) ARGF14
ARCON
SMOVL C00714 BC00714 V=10.0  +MOVJ EC00714
ARCOF
SMOVL C00715 BC00715 V=400.0  +MOVJ EC00715
SMOVL C00716 BC00716 V=1000.0  +MOVJ EC00716
SFTOF3D
SMOVL C00717 BC00717 V=400.0  +MOVJ EC00717
SFTON3D P027
MACRO1 MJ#(0) ARGF9
SMOVL C00718 BC00718 V=150.0 PL=0  +MOVJ EC00718
ARCON
SFTON3D P026
SMOVL C00719 BC00719 V=11.7  +MOVJ EC00719
SMOVC C00720 BC00720 V=13.3  +MOVJ EC00720
SMOVC C00721 BC00721 V=13.3  +MOVJ EC00721
SMOVC C00722 BC00722 V=13.3  +MOVJ EC00722
SFTON3D P027
SMOVL C00723 BC00723 V=11.7  +MOVJ EC00723
SMOVL C00724 BC00724 V=11.7  +MOVJ EC00724
SMOVC C00725 BC00725 V=13.3  +MOVJ EC00725
SMOVC C00726 BC00726 V=13.3  +MOVJ EC00726
SMOVC C00727 BC00727 V=13.3  +MOVJ EC00727
ARCOF
SMOVL C00728 BC00728 V=333.3  +MOVJ EC00728
SFTOF3D
SMOVL C00729 BC00729 V=400.0  +MOVJ EC00729
SFTON3D P025
MACRO1 MJ#(0) ARGF9
SMOVL C00730 BC00730 V=150.0 PL=0  +MOVJ EC00730
ARCON
SFTON3D P024
SMOVL C00731 BC00731 V=11.7  +MOVJ EC00731
SMOVC C00732 BC00732 V=13.3  +MOVJ EC00732
SMOVC C00733 BC00733 V=13.3  +MOVJ EC00733
SMOVC C00734 BC00734 V=13.3  +MOVJ EC00734
SFTON3D P025
SMOVL C00735 BC00735 V=11.7  +MOVJ EC00735
SMOVL C00736 BC00736 V=11.7  +MOVJ EC00736
SMOVC C00737 BC00737 V=13.3  +MOVJ EC00737
SMOVC C00738 BC00738 V=13.3  +MOVJ EC00738
SMOVC C00739 BC00739 V=13.3  +MOVJ EC00739
ARCOF
SMOVL C00740 BC00740 V=333.3  +MOVJ EC00740
SFTOF3D
SMOVL C00741 BC00741 V=666.7  +MOVJ EC00741
MOVJ C00742 BC00742 VJ=100.00  +MOVJ EC00742 VJ=100.00
MOVJ C00743 BC00743 VJ=100.00  +MOVJ EC00743 VJ=100.00
'6
'Path W1895
SFTOF3D
SFTON3D P022
MOVJ C00744 BC00744 VJ=40.00  +MOVJ EC00744 VJ=100.00
SMOVL C00745 BC00745 V=400.0  +MOVJ EC00745
SMOVL C00746 BC00746 V=133.3 PL=0  +MOVJ EC00746
SREFP 1 C00747 BC00747  +REFP EC00747
SREFP 2 C00748 BC00748  +REFP EC00748
MACRO1 MJ#(0) ARGF14
ARCON
SMOVL C00749 BC00749 V=11.7  +MOVJ EC00749
ARCOF
SMOVL C00750 BC00750 V=166.7  +MOVJ EC00750
SMOVL C00751 BC00751 V=166.7  +MOVJ EC00751
SMOVL C00752 BC00752 V=166.7 PL=0  +MOVJ EC00752
ARCON
SMOVL C00753 BC00753 V=11.7  +MOVJ EC00753
ARCOF
SMOVL C00754 BC00754 V=400.0  +MOVJ EC00754
SMOVL C00755 BC00755 V=1000.0  +MOVJ EC00755
SFTOF3D
MOVJ C00756 BC00756 VJ=100.00  +MOVJ EC00756 VJ=100.00
'Path W1896
SFTOF3D
SFTON3D P022
MOVJ C00757 BC00757 VJ=50.00  +MOVJ EC00757 VJ=100.00
SMOVL C00758 BC00758 V=400.0  +MOVJ EC00758
SMOVL C00759 BC00759 V=133.3 PL=0  +MOVJ EC00759
SREFP 1 C00760 BC00760  +REFP EC00760
SREFP 2 C00761 BC00761  +REFP EC00761
MACRO1 MJ#(0) ARGF14
ARCON
SMOVL C00762 BC00762 V=12.5  +MOVJ EC00762
ARCOF
SMOVL C00763 BC00763 V=400.0  +MOVJ EC00763
SMOVL C00764 BC00764 V=1000.0  +MOVJ EC00764
SFTOF3D
'7
'Path W1897
SFTOF3D
SFTON3D P022
MOVJ C00765 BC00765 VJ=100.00  +MOVJ EC00765 VJ=100.00
SMOVL C00766 BC00766 V=400.0  +MOVJ EC00766
SMOVL C00767 BC00767 V=133.3 PL=0  +MOVJ EC00767
SREFP 1 C00768 BC00768  +REFP EC00768
SREFP 2 C00769 BC00769  +REFP EC00769
MACRO1 MJ#(0) ARGF14
ARCON
SMOVL C00770 BC00770 V=12.5  +MOVJ EC00770
ARCOF
SMOVL C00771 BC00771 V=400.0  +MOVJ EC00771
SMOVL C00772 BC00772 V=1000.0  +MOVJ EC00772
SMOVL C00773 BC00773 V=1000.0  +MOVJ EC00773
SFTOF3D
MOVJ C00774 BC00774 VJ=100.00  +MOVJ EC00774 VJ=100.00
'Path W1898
SFTOF3D
SFTON3D P022
MOVJ C00775 BC00775 VJ=100.00  +MOVJ EC00775 VJ=100.00
SMOVL C00776 BC00776 V=400.0  +MOVJ EC00776
SMOVL C00777 BC00777 V=133.3 PL=0  +MOVJ EC00777
SREFP 1 C00778 BC00778  +REFP EC00778
SREFP 2 C00779 BC00779  +REFP EC00779
MACRO1 MJ#(0) ARGF14
ARCON
SMOVL C00780 BC00780 V=12.5  +MOVJ EC00780
ARCOF
SMOVL C00781 BC00781 V=400.0  +MOVJ EC00781
SMOVL C00782 BC00782 V=1000.0  +MOVJ EC00782
SFTOF3D
MOVJ C00783 BC00783 VJ=100.00  +MOVJ EC00783 VJ=20.00
MOVJ C00784 BC00784 VJ=100.00  +MOVJ EC00784 VJ=20.00
MOVJ C00785 BC00785 VJ=100.00  +MOVJ EC00785 VJ=20.00
MOVJ C00786 BC00786 VJ=100.00  +MOVJ EC00786 VJ=100.00
MOVL C00787 BC00787 V=666.7  +MOVJ EC00787 VJ=100.00
SFTON3D P028
MOVL C00788 BC00788 V=666.7  +MOVJ EC00788 VJ=100.00
MACRO1 MJ#(0) ARGF9
SMOVL C00789 BC00789 V=166.7 PL=0  +MOVJ EC00789
ARCON
SMOVL C00790 BC00790 V=13.3  +MOVJ EC00790
SFTON3D P029
SMOVL C00791 BC00791 V=13.3  +MOVJ EC00791
SMOVL C00792 BC00792 V=13.3  +MOVJ EC00792
SMOVL C00793 BC00793 V=13.3  +MOVJ EC00793
SMOVL C00794 BC00794 V=13.3  +MOVJ EC00794
ARCOF
SMOVL C00795 BC00795 V=666.7  +MOVJ EC00795
SFTOF3D
SMOVL C00796 BC00796 V=666.7  +MOVJ EC00796
MOVJ C00797 BC00797 VJ=100.00  +MOVJ EC00797 VJ=100.00
MOVJ C00798 BC00798 VJ=100.00  +MOVJ EC00798 VJ=20.00
MOVJ C00799 BC00799 VJ=100.00  +MOVJ EC00799 VJ=100.00
SFTOF3D
END
